TYPE ST_CSL_Diagnostic :
STRUCT
	(*
	aCritical 	: 	ARRAY[0..GVL_Diagnostic.cMAXEVENTS - 1] OF BOOL; 		// critic events   
	aError 		: 	ARRAY[0..GVL_Diagnostic.cMAXEVENTS - 1] OF BOOL; 		// errors    
	aWarning 	: 	ARRAY[0..GVL_Diagnostic.cMAXEVENTS - 1] OF BOOL; 	 	// reports    
	aInfo 		: 	ARRAY[0..GVL_Diagnostic.cMAXEVENTS - 1] OF BOOL; 		// informations   
 	aVerbose 	: 	ARRAY[0..GVL_Diagnostic.cMAXEVENTS - 1] OF BOOL;  		// message
*)
END_STRUCT
END_TYPE

(* stored: Version 1.1.0.1, ProductVersion 3.1.4024.12
   DUT ST_CSL_Diagnostic: Id {2496aee4-be2f-4bf2-9b51-08798cf085f2} *)
